// SIMATIC S7-200 project (STEP 7-Micro/WIN), CPU 222 REL 01.22

ORGANIZATION_BLOCK PRINCIPAL:OB1
TITLE=COMENTARIOS DEL PROGRAMA
BEGIN
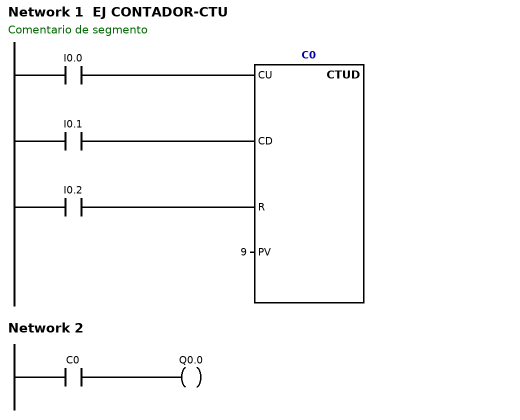
Network 1 // EJ CONTADOR-CTU

// Comentario de segmento
// (network saved uncompiled; LAD cells follow)
// row 0: c0 -| |- I0.0  c1 --  c2 [CTUD C0 CU:=power@row0, CD:=power@row1, R:=power@row2, PV:=9]
// row 1: c0 -| |- I0.1  c1 --  c2 [box]
// row 2: c0 -| |- I0.2  c1 --  c2 [box]
// row 3: c2 [box]
Network 2
LD     C0
=      Q0.0
END_ORGANIZATION_BLOCK
